TYPE
    E_TalkToGateway_Err :
    (
        e_NoIPAddress           := 10,
        e_NoPortNumber          := 20,
        e_NoDeviceID            := 30,
        e_DeviceIDOutsideLimits := 31,
        e_DeviceIDNotFound      := 32,
		e_JSONRequestError		:= 40
        );
END_TYPE

(* stored: Version 1.1.0.1, ProductVersion 3.1.4024.15
   DUT E_TalkToGateway_Err: Id {635f7ad4-042c-41e7-bd5f-1e19928fc21b} *)
